(* CODESYS project MyPCEtherCAT_2ESC.project

Project tree, tasks and I/O mapping:
  Device : CODESYS Control Win V3, 3S - Smart Software Solutions GmbH, order no. 305021, version 3.5.10.0
    application MotorControl
      libraries: Standard, * (System)
      task MainTask (cyclic, interval 4 ms, priority 0) calls PLC_PRG
      task ETH (cyclic, interval 4 ms, priority 0) calls EtherCAT_Master.EtherCAT_Task
      program PLC_PRG [LD]
    EtherCAT_Master : EtherCAT Master, 3S - Smart Software Solutions GmbH, version 3.5.10.0
        settings: NetworkName = 'Připojení k místní síti'; NetworkName = "Připojení k místní síti"; SrcAddress1 = 64533; SrcAddress2 = 3035404439
      XMC_ESC : XMC_ESC, Bahoza, order no. XMC_ESC, version Revision=16#00000000
          settings: EnableExpertSettings = True; StationAlias = 0; DC sync0 cycletime = 4000; DC sync1 cycletime = 4000
          input  BTN_ON : BIT  // IN_GEN_Bit1
          input  BTN_OFF : BIT  // IN_GEN_Bit2
          unmapped channels: OUT_GEN_INT1, OUT_GEN_INT2, OUT_GEN_INT3, OUT_GEN_INT4, OUT_GEN_Bit1, OUT_GEN_Bit2, OUT_GEN_Bit3, OUT_GEN_Bit4, OUT_GEN_Bit5, OUT_GEN_Bit6, OUT_GEN_Bit7, OUT_GEN_Bit8, IN_GEN_INT1, IN_GEN_INT2, IN_GEN_INT3, IN_GEN_INT4, IN_GEN_Bit3, IN_GEN_Bit4, IN_GEN_Bit5, IN_GEN_Bit6, IN_GEN_Bit7, IN_GEN_Bit8
      XMC_ESC_1 : XMC_ESC, Bahoza, order no. XMC_ESC, version Revision=16#00000000
          settings: EnableExpertSettings = True; StationAlias = 0; DC sync0 cycletime = 4000; DC sync1 cycletime = 4000
          output MOTOR_ON : BIT  // OUT_GEN_Bit1
          unmapped channels: OUT_GEN_INT1, OUT_GEN_INT2, OUT_GEN_INT3, OUT_GEN_INT4, OUT_GEN_Bit2, OUT_GEN_Bit3, OUT_GEN_Bit4, OUT_GEN_Bit5, OUT_GEN_Bit6, OUT_GEN_Bit7, OUT_GEN_Bit8, IN_GEN_INT1, IN_GEN_INT2, IN_GEN_INT3, IN_GEN_INT4, IN_GEN_Bit1, IN_GEN_Bit2, IN_GEN_Bit3, IN_GEN_Bit4, IN_GEN_Bit5, IN_GEN_Bit6, IN_GEN_Bit7, IN_GEN_Bit8
*)

// Device/MotorControl/PLC_PRG
PROGRAM PLC_PRG
VAR
END_VAR

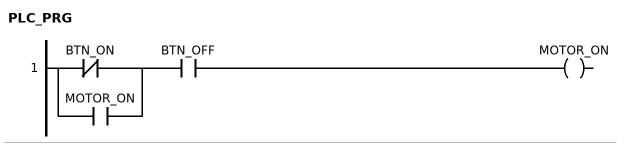
// NETWORK 1
MOTOR_ON := (NOT BTN_ON OR MOTOR_ON) AND BTN_OFF;

END_PROGRAM
